{attribute 'GeneratedUsingTerminal: EL3632-0000-0022'}
{attribute addProperty BoxType "EL3632-0000-0022"}
{attribute addProperty Id "Ch1_StatusAT %I*Ch1_Status_758244858Ch1_Sample_0AT %I*Ch1_Sample_A71DD5012Ch1_Sample_1AT %I*Ch1_Sample_A71DD5012Ch1_Sample_2AT %I*Ch1_Sample_A71DD5012Ch1_Sample_3AT %I*Ch1_Sample_A71DD5012Ch1_Sample_4AT %I*Ch1_Sample_A71DD5012Ch1_Sample_5AT %I*Ch1_Sample_A71DD5012Ch1_Sample_6AT %I*Ch1_Sample_A71DD5012Ch1_Sample_7AT %I*Ch1_Sample_A71DD5012Ch1_Sample_8AT %I*Ch1_Sample_A71DD5012Ch1_Sample_9AT %I*Ch1_Sample_A71DD5012Ch2_StatusAT %I*Ch2_Status_758244858Ch2_Sample_0AT %I*Ch2_Sample_9F6886E62Ch2_Sample_1AT %I*Ch2_Sample_9F6886E62Ch2_Sample_2AT %I*Ch2_Sample_9F6886E62Ch2_Sample_3AT %I*Ch2_Sample_9F6886E62Ch2_Sample_4AT %I*Ch2_Sample_9F6886E62Ch2_Sample_5AT %I*Ch2_Sample_9F6886E62Ch2_Sample_6AT %I*Ch2_Sample_9F6886E62Ch2_Sample_7AT %I*Ch2_Sample_9F6886E62Ch2_Sample_8AT %I*Ch2_Sample_9F6886E62Ch2_Sample_9AT %I*Ch2_Sample_9F6886E62NextSync1TimeAT %I*NextSync1Time_9AFDC2758Sample_CountAT %I*Sample_Count_EA88CAD92WcStateAT %I*WcState_9091E0EB2InfoDataAT %I*InfoData_1088C70510"}
{attribute addProperty CRC "1809965612"}
{attribute addProperty Size "78"}
TYPE EL3632_6BE1E22C EXTENDS EtcSlaveTerminalBase_947E5A46 :
STRUCT
	{attribute addProperty Name "Ch1_Status"}
	Ch1_Status : Ch1_Status_75824485;
	{attribute addProperty Name "Ch1_Sample_0"}
	Ch1_Sample_0 : Ch1_Sample_A71DD501;
	{attribute addProperty Name "Ch1_Sample_1"}
	Ch1_Sample_1 : Ch1_Sample_A71DD501;
	{attribute addProperty Name "Ch1_Sample_2"}
	Ch1_Sample_2 : Ch1_Sample_A71DD501;
	{attribute addProperty Name "Ch1_Sample_3"}
	Ch1_Sample_3 : Ch1_Sample_A71DD501;
	{attribute addProperty Name "Ch1_Sample_4"}
	Ch1_Sample_4 : Ch1_Sample_A71DD501;
	{attribute addProperty Name "Ch1_Sample_5"}
	Ch1_Sample_5 : Ch1_Sample_A71DD501;
	{attribute addProperty Name "Ch1_Sample_6"}
	Ch1_Sample_6 : Ch1_Sample_A71DD501;
	{attribute addProperty Name "Ch1_Sample_7"}
	Ch1_Sample_7 : Ch1_Sample_A71DD501;
	{attribute addProperty Name "Ch1_Sample_8"}
	Ch1_Sample_8 : Ch1_Sample_A71DD501;
	{attribute addProperty Name "Ch1_Sample_9"}
	Ch1_Sample_9 : Ch1_Sample_A71DD501;
	{attribute addProperty Name "Ch2_Status"}
	Ch2_Status : Ch2_Status_75824485;
	{attribute addProperty Name "Ch2_Sample_0"}
	Ch2_Sample_0 : Ch2_Sample_9F6886E6;
	{attribute addProperty Name "Ch2_Sample_1"}
	Ch2_Sample_1 : Ch2_Sample_9F6886E6;
	{attribute addProperty Name "Ch2_Sample_2"}
	Ch2_Sample_2 : Ch2_Sample_9F6886E6;
	{attribute addProperty Name "Ch2_Sample_3"}
	Ch2_Sample_3 : Ch2_Sample_9F6886E6;
	{attribute addProperty Name "Ch2_Sample_4"}
	Ch2_Sample_4 : Ch2_Sample_9F6886E6;
	{attribute addProperty Name "Ch2_Sample_5"}
	Ch2_Sample_5 : Ch2_Sample_9F6886E6;
	{attribute addProperty Name "Ch2_Sample_6"}
	Ch2_Sample_6 : Ch2_Sample_9F6886E6;
	{attribute addProperty Name "Ch2_Sample_7"}
	Ch2_Sample_7 : Ch2_Sample_9F6886E6;
	{attribute addProperty Name "Ch2_Sample_8"}
	Ch2_Sample_8 : Ch2_Sample_9F6886E6;
	{attribute addProperty Name "Ch2_Sample_9"}
	Ch2_Sample_9 : Ch2_Sample_9F6886E6;
	{attribute addProperty Name "NextSync1Time"}
	NextSync1Time : NextSync1Time_9AFDC275;
	{attribute addProperty Name "Sample_Count"}
	Sample_Count : Sample_Count_EA88CAD9;
	{attribute addProperty Name "WcState"}
	WcState : WcState_9091E0EB;
	{attribute addProperty Name "InfoData"}
	InfoData : InfoData_1088C705;
END_STRUCT
END_TYPE

(* stored: Version 1.2.0.0, ProductVersion 3.1.4024.9
   DUT EL3632_6BE1E22C: Id {4771cf96-a9ef-4215-a56d-7615a258618f} *)
